KUKA KRL program: SET_MAXFORCE.src

&ACCESS RV
&REL 3
&PARAM TEMPLATE = C:\KRC\Roboter\Template\FunctionVorgabe
&PARAM EDITMASK = *
DEFFCT BOOL SET_MAXFORCE( X_VAL:IN, Y_VAL:IN, Z_VAL:IN, A_VAL:IN, B_VAL:IN, C_VAL:IN)

REAL X_VAL, Y_VAL, Z_VAL
REAL A_VAL, B_VAL, C_VAL

$STIFFNESS.MAXFORCE.X = X_VAL
$STIFFNESS.MAXFORCE.Y = Y_VAL
$STIFFNESS.MAXFORCE.Z = Z_VAL
$STIFFNESS.MAXFORCE.A = A_VAL
$STIFFNESS.MAXFORCE.B = B_VAL
$STIFFNESS.MAXFORCE.C = C_VAL

$STIFFNESS.COMMIT = TRUE

RETURN TRUE

ENDFCT
